// TIA Portal V20 export
// export: Created 2026-07-10T11:12:27.1506588Z, ExportSetting WithDefaults, DisplayName Totally Integrated Automation Portal, DisplayVersion V20, DisplayName TIA Portal Openness, DisplayVersion V20, DisplayName TIA Portal Version Control Interface, DisplayVersion V20, DisplayName STEP 7 Professional, DisplayVersion V20, DisplayName STEP 7 Safety, DisplayVersion V20, DisplayName WinCC Basic/Comfort/Advanced, DisplayVersion V20, DisplayName WinCC Unified, DisplayVersion V20
DATA_BLOCK "WorkModeCycle_DB"   // DB3
VERSION : 0.1
// stored: AutoNumber true, DBAccessibleFromOPCUA true, InstanceOfName WorkModeCycle, InstanceOfType FB
"WorkModeCycle"
   // VAR
   //    "step" : Int;
   //    tod : Time_Of_Day;
   //    "return" : Int;
   //    dtl : DTL;
   //    "time" : Time;
   //    fracDay : Real;
   // END_VAR
BEGIN
END_DATA_BLOCK
